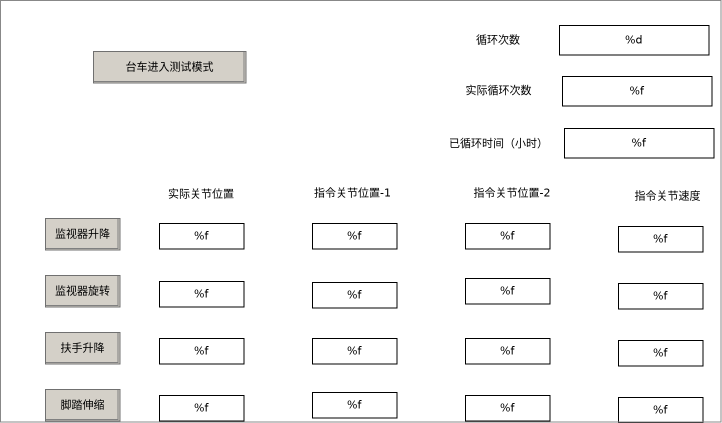
VISUALIZATION cartCycleTest  // 722x423
    Button (93,51 153x32), "台车进入测试模式", colour toggle: g_cycleTest.m_carEnterCycleTest
        toggle g_cycleTest.m_carEnterCycleTest
    Rectangle (559,25 150x30), "%d", text variable: g_cycleTest.m_targetCycleNumCar
        OnMouseClick: write the text variable via Default
    Label (456,25 84x30), "循环次数"
    Label (293,179 119x28), "指令关节位置-1"
    Label (151,179 100x30), "实际关节位置"
    Rectangle (159,395 85x26), "%f", text variable: g_systemInfo.m_cartJntInfo[4].m_curJntPos
    Rectangle (159,223 85x26), "%f", text variable: g_systemInfo.m_cartJntInfo[1].m_curJntPos
    Rectangle (159,281 85x26), "%f", text variable: g_systemInfo.m_cartJntInfo[2].m_curJntPos
    Rectangle (159,338 85x26), "%f", text variable: g_systemInfo.m_cartJntInfo[3].m_curJntPos
    Rectangle (312,223 85x26), "%f", text variable: g_cycleTest.m_targetJntPosCar[1][1]
        OnMouseClick: write the text variable via Default
    Rectangle (312,282 85x26), "%f", text variable: g_cycleTest.m_targetJntPosCar[1][2]
        OnMouseClick: write the text variable via Default
    Rectangle (312,338 85x26), "%f", text variable: g_cycleTest.m_targetJntPosCar[1][3]
        OnMouseClick: write the text variable via Default
    Rectangle (312,392 85x26), "%f", text variable: g_cycleTest.m_targetJntPosCar[1][4]
        OnMouseClick: write the text variable via Default
    Label (454,179 116x28), "指令关节位置-2"
    Rectangle (465,223 85x26), "%f", text variable: g_cycleTest.m_targetJntPosCar[2][1]
        OnMouseClick: write the text variable via Default
    Rectangle (465,278 85x26), "%f", text variable: g_cycleTest.m_targetJntPosCar[2][2]
        OnMouseClick: write the text variable via Default
    Rectangle (465,338 85x26), "%f", text variable: g_cycleTest.m_targetJntPosCar[2][3]
        OnMouseClick: write the text variable via Default
    Rectangle (465,395 85x26), "%f", text variable: g_cycleTest.m_targetJntPosCar[2][4]
        OnMouseClick: write the text variable via Default
    Label (613,182 109x28), "指令关节速度"
    Rectangle (618,226 85x26), "%f", text variable: g_cycleTest.m_targetJntVelCar[1]
        OnMouseClick: write the text variable via Default
    Rectangle (618,283 85x26), "%f", text variable: g_cycleTest.m_targetJntVelCar[2]
        OnMouseClick: write the text variable via Default
    Rectangle (618,340 85x26), "%f", text variable: g_cycleTest.m_targetJntVelCar[3]
        OnMouseClick: write the text variable via Default
    Rectangle (618,397 85x26), "%f", text variable: g_cycleTest.m_targetJntVelCar[4]
        OnMouseClick: write the text variable via Default
    Rectangle (562,76 150x30), "%f", text variable: g_cycleTest.m_curCycleNumCar
        OnMouseClick: write the text variable via Default
    Label (450,80 97x21), "实际循环次数"
    Rectangle (564,128 150x30), "%f", text variable: g_cycleTest.m_curCycleTimeCar
        OnMouseClick: write the text variable via Default
    Label (438,133 121x21), "已循环时间（小时）"
    Button (45,218 75x32), "监视器升降", colour toggle: g_motionTest.m_jntEnableCar[1]
        toggle g_motionTest.m_jntEnableCar[1]
    Button (45,275 75x32), "监视器旋转", colour toggle: g_motionTest.m_jntEnableCar[2]
        toggle g_motionTest.m_jntEnableCar[2]
    Button (45,332 75x32), "扶手升降", colour toggle: g_motionTest.m_jntEnableCar[3]
        toggle g_motionTest.m_jntEnableCar[3]
    Button (45,389 75x32), "脚踏伸缩", colour toggle: g_motionTest.m_jntEnableCar[4]
        toggle g_motionTest.m_jntEnableCar[4]
END_VISUALIZATION

(* stored: Version 1.1.0.1, ProductVersion 3.1.4024.11
   Visu cartCycleTest: Id {3908e9c4-c2cf-4ad1-b2e8-0e1877b11c30} *)
